{attribute 'qualified_only'}
{attribute 'strict'}
TYPE EN_TempControlMode :
(
	TEMP_MODE_MANUAL := 1,
	TEMP_MODE_HEATCOOL,
	TEMP_MODE_STERI
);
END_TYPE

(* stored: Version 1.1.0.1, ProductVersion 3.1.4022.7
   DUT EN_TempControlMode: Id {eccf7990-447d-43f4-82f3-08b6b112ba01} *)
